// TwinCAT 3 PLC project SampleLibraryA
// Title: SampleLibraryA
// Company: blark-testing
// ProjectVersion: 1.0.0
// ProgramVersion: 3.1.4022.7
// libraries:
//   Tc2_Standard, * (Beckhoff Automation GmbH)
//   Tc2_System, * (Beckhoff Automation GmbH)
//   Tc3_Module, * (Beckhoff Automation GmbH)
// project tree:
//   POUs/ FB_SampleA_Test.TcPOU
// real-time tasks:
//   TASK PlcTask: cycle T#10ms, priority 20, ADS port 350

// ---- POUs/FB_SampleA_Test.TcPOU
FUNCTION_BLOCK FB_SampleA_Test
VAR_INPUT
	{attribute 'pytmc' := '
		pv: fInput
		io: io
	'}
	fInput : LREAL;
END_VAR
VAR_OUTPUT
	{attribute 'pytmc' := '
		pv: fOutput
		io: input
	'}
	fOutput : LREAL;
END_VAR
VAR
END_VAR

fOutput := fInput;

END_FUNCTION_BLOCK
